{attribute addProperty BoxType "ER2038-0001-0017"}
{attribute addProperty Id "Diag_ChannelAT %I*ARRAY[0..7] OF Diag_Channel_E4AEF59E6480ChannelAT %Q*ARRAY[0..7] OF Channel_7F374EB06480WcStateAT %I*WcState_98A4DF7520.250InfoDataAT %I*InfoData_192954DE1620"}
{attribute addProperty CRC "1245809967"}
{attribute addProperty SizeInBites "146"}
{attribute addProperty SizeInBytes "18.25"}
TYPE ER2038_9444C9D3 :
STRUCT
	{attribute addProperty Name "Diag_Channel"}
	Diag_Channel : ARRAY[0..7] OF Diag_Channel_E4AEF59E;
	{attribute addProperty Name "Channel"}
	Channel : ARRAY[0..7] OF Channel_7F374EB0;
	{attribute addProperty Name "WcState"}
	WcState : WcState_98A4DF75;
	{attribute addProperty Name "InfoData"}
	InfoData : InfoData_192954DE;
END_STRUCT
END_TYPE

(* stored: Version 1.2.0.0, ProductVersion 3.1.4024.9
   DUT ER2038_9444C9D3: Id {de9be61e-648c-4171-abaa-075a41e14903} *)
